(* Logix 5000 project; controller EuniceF_ICA01 vendor 1 type 14 code 150 rev 37.11; software revision 37.00 *)

TASK MainTask (continuous, watchdog 500 ms) : MainProgram

MODULES
   Local : vendor 1 type 14 code 150 (Compact 0, rev 37.11)
      Discrete_IO : Embedded (Compact 1, rev 3.1, Output RPI 20 ms)
      Analog_IO : Embedded (Compact 2, rev 1.1, Output RPI 80 ms)
      Counters : Embedded (Compact 3, rev 1.1, Output RPI 20 ms)
END_MODULES

VAR_GLOBAL   (* controller tags *)
   Light_1 : ALIAS FOR Local:1:O.Data.1;
   Light_2 : ALIAS FOR Local:1:O.Data.2;
   SW1 : ALIAS FOR Local:1:I.Data.11;
   SW2 : ALIAS FOR Local:1:I.Data.12;
   SW3 : ALIAS FOR Local:1:I.Data.8;
   SW4 : ALIAS FOR Local:1:I.Data.9;
END_VAR

PROGRAM MainProgram   (* main routine MainRoutine *)

ROUTINE MainRoutine   (* ladder *)
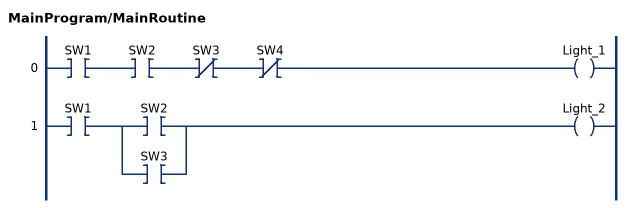
   0: XIC(SW1)XIC(SW2)XIO(SW3)XIO(SW4)OTE(Light_1);
   1: XIC(SW1)[XIC(SW2) ,XIC(SW3) ]OTE(Light_2);
END_ROUTINE
END_PROGRAM
